TYPE "IPC_Msg_Log_MES"
VERSION : 0.1
// Block: IPC_Msg_Log_MES
   STRUCT
      Id : DInt;
      timestamp : String;
      topic : UDInt;
      payLoad_1 : String;
      payLoad_2 : String;
   END_STRUCT;

END_TYPE
